(* IEC 61131-3 sources: plc_generation_empirical_study/datasets/task_bank_v0_3/tasks/C01_B07_composite, 2 files *)

(* ---- interface.st ---- *)
FUNCTION_BLOCK C01_B07_composite
VAR_INPUT
    A_ChA : BOOL;
    A_ChB : BOOL;
    A_TestMode : BOOL;
    A_TestPermit : BOOL;
    A_ProcessRequest : BOOL;
    B_AutoMode : BOOL;
    B_AutoDemand : BOOL;
    B_ManualDemand : BOOL;
    B_SafetyOK : BOOL;
    B_Inhibit : BOOL;
    SubsystemBEnable : BOOL;
    CrossReset : BOOL;
END_VAR
VAR_OUTPUT
    A_SafeEnable : BOOL;
    A_Disagree : BOOL;
    A_TestActive : BOOL;
    B_Command : BOOL;
    B_Blocked : BOOL;
    CrossReady : BOOL;
    CrossBlocked : BOOL;
END_VAR
END_FUNCTION_BLOCK

(* ---- reference.st ---- *)
FUNCTION_BLOCK C01_B07_composite
VAR_INPUT
    A_ChA : BOOL;
    A_ChB : BOOL;
    A_TestMode : BOOL;
    A_TestPermit : BOOL;
    A_ProcessRequest : BOOL;
    B_AutoMode : BOOL;
    B_AutoDemand : BOOL;
    B_ManualDemand : BOOL;
    B_SafetyOK : BOOL;
    B_Inhibit : BOOL;
    SubsystemBEnable : BOOL;
    CrossReset : BOOL;
END_VAR
VAR_OUTPUT
    A_SafeEnable : BOOL;
    A_Disagree : BOOL;
    A_TestActive : BOOL;
    B_Command : BOOL;
    B_Blocked : BOOL;
    CrossReady : BOOL;
    CrossBlocked : BOOL;
END_VAR

A_Disagree := A_ChA <> A_ChB;
A_TestActive := A_TestMode AND A_TestPermit;
IF A_TestMode THEN
    A_SafeEnable := A_ProcessRequest AND A_TestPermit AND A_ChA;
ELSE
    A_SafeEnable := A_ProcessRequest AND A_ChA AND A_ChB;
END_IF;

IF CrossReset THEN
    CrossReady := FALSE;
ELSIF A_SafeEnable THEN
    CrossReady := TRUE;
END_IF;
CrossBlocked := SubsystemBEnable AND (NOT CrossReady);

IF SubsystemBEnable AND CrossReady THEN
    B_Command := ((B_AutoMode AND B_AutoDemand) OR ((NOT B_AutoMode) AND B_ManualDemand))
               AND B_SafetyOK AND (NOT B_Inhibit);
    B_Blocked := ((B_AutoMode AND B_AutoDemand) OR ((NOT B_AutoMode) AND B_ManualDemand))
               AND ((NOT B_SafetyOK) OR B_Inhibit);
ELSE
    B_Command := FALSE;
    B_Blocked := FALSE;
END_IF;

END_FUNCTION_BLOCK
